% RSLogix 500 project DIGITAL_CONTROL_LOGIC.RSS, saved by version 8.30.00.16 %
PROJECT "DCL_L2P1"    % processor: Bul.1763 MicroLogix 1100 Series B %

PROGRAM FILES
  LAD 2 "MAIN"  5 rungs
  LAD 3 "DIGI IN"  3 rungs
  LAD 4 "DIGI OUT"  3 rungs
  LAD 5 "CONTROL"  7 rungs

DATA FILES
  O0 OUTPUT  5 elements
  I1 INPUT  7 elements
  S2 STATUS  66 elements
  B3 BINARY  3 elements
  T4 TIMER  4 elements
  C5 COUNTER  1 elements
  R6 CONTROL  1 elements
  N7 INTEGER  2 elements
  F8 FLOAT  1 elements

LADDER 2 "MAIN"
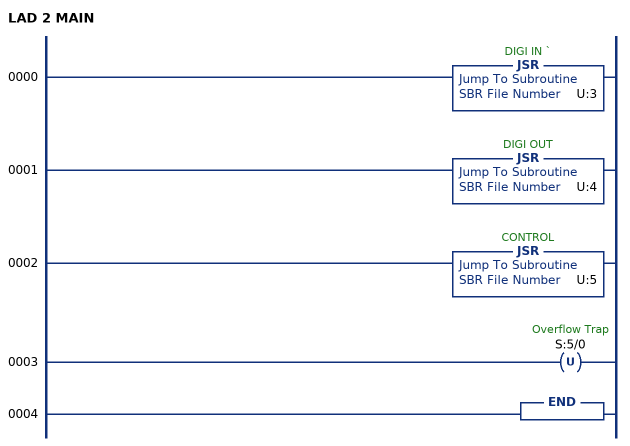
% Rung: 0 %
SOR JSR U:3 EOR
%   U:3  "DIGI IN `" %
% Rung: 1 %
SOR JSR U:4 EOR
%   U:4  "DIGI OUT" %
% Rung: 2 %
SOR JSR U:5 EOR
%   U:5  "CONTROL" %
% Rung: 3 %
SOR OTU S:5/0 EOR
%   S:5/0  "Overflow Trap" %
% Rung: 4 %
SOR END EOR

LADDER 3 "DIGI IN"
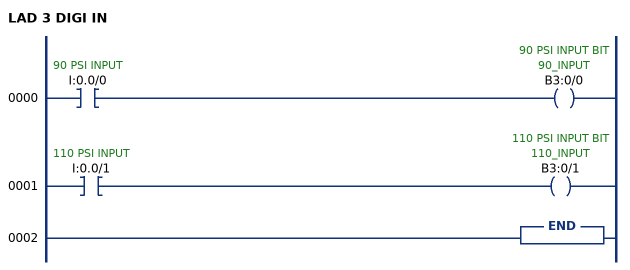
% Rung: 0 %
SOR XIC I:0.0/0 OTE B3:0/0 EOR
%   I:0.0/0  "90 PSI INPUT" %
%   B3:0/0  90_INPUT  "90 PSI INPUT BIT" %
% Rung: 1 %
SOR XIC I:0.0/1 OTE B3:0/1 EOR
%   I:0.0/1  "110 PSI INPUT" %
%   B3:0/1  110_INPUT  "110 PSI INPUT BIT" %
% Rung: 2 %
SOR END EOR

LADDER 4 "DIGI OUT"
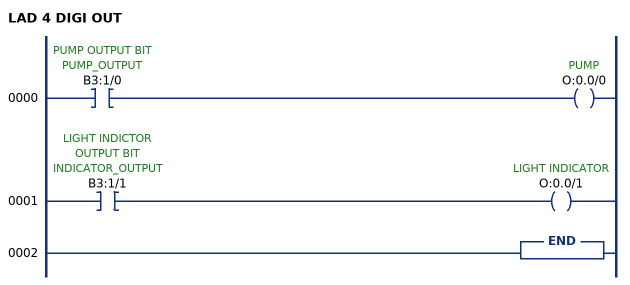
% Rung: 0 %
SOR XIC B3:1/0 OTE O:0.0/0 EOR
%   B3:1/0  PUMP_OUTPUT  "PUMP OUTPUT BIT" %
%   O:0.0/0  "PUMP" %
% Rung: 1 %
SOR XIC B3:1/1 OTE O:0.0/1 EOR
%   B3:1/1  INDICATOR_OUTPUT  "LIGHT INDICTOR OUTPUT BIT" %
%   O:0.0/1  "LIGHT INDICATOR" %
% Rung: 2 %
SOR END EOR

LADDER 5 "CONTROL"
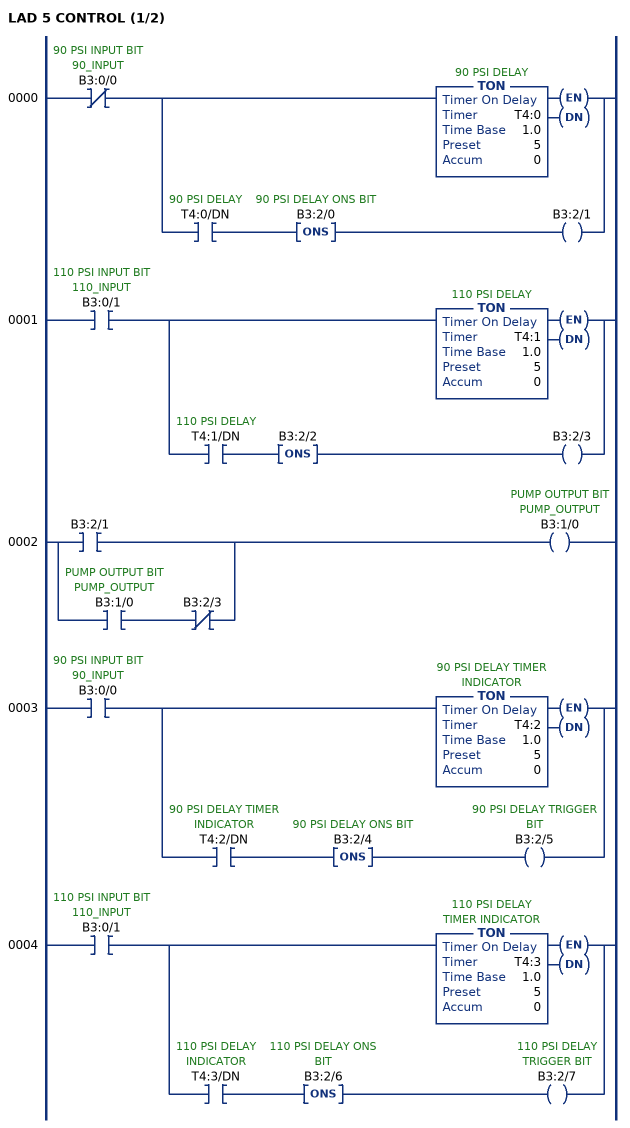
% Rung: 0 %
SOR XIO B3:0/0 BST TON T4:0 1.0 5 0 NXB XIC T4:0/DN ONS B3:2/0 OTE B3:2/1 BND EOR
%   B3:0/0  90_INPUT  "90 PSI INPUT BIT" %
%   T4:0  "90 PSI DELAY" %
%   T4:0/DN  "90 PSI DELAY" %
%   B3:2/0  "90 PSI DELAY ONS BIT" %
% Rung: 1 %
SOR XIC B3:0/1 BST TON T4:1 1.0 5 0 NXB XIC T4:1/DN ONS B3:2/2 OTE B3:2/3 BND EOR
%   B3:0/1  110_INPUT  "110 PSI INPUT BIT" %
%   T4:1  "110 PSI DELAY" %
% Rung: 2 %
SOR BST XIC B3:2/1 NXB XIC B3:1/0 XIO B3:2/3 BND OTE B3:1/0 EOR
%   B3:1/0  PUMP_OUTPUT  "PUMP OUTPUT BIT" %
% Rung: 3 %
SOR XIC B3:0/0 BST TON T4:2 1.0 5 0 NXB XIC T4:2/DN ONS B3:2/4 OTE B3:2/5 BND EOR
%   B3:0/0  90_INPUT  "90 PSI INPUT BIT" %
%   T4:2  "90 PSI DELAY TIMER INDICATOR" %
%   B3:2/4  "90 PSI DELAY ONS BIT" %
%   B3:2/5  "90 PSI DELAY TRIGGER BIT" %
% Rung: 4 %
SOR XIC B3:0/1 BST TON T4:3 1.0 5 0 NXB XIC T4:3/DN ONS B3:2/6 OTE B3:2/7 BND EOR
%   B3:0/1  110_INPUT  "110 PSI INPUT BIT" %
%   T4:3  "110 PSI DELAY TIMER INDICATOR" %
%   T4:3/DN  "110 PSI DELAY INDICATOR" %
%   B3:2/6  "110 PSI DELAY ONS BIT" %
%   B3:2/7  "110 PSI DELAY TRIGGER BIT" %

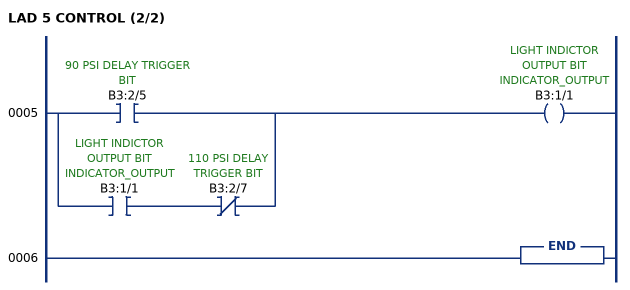
% Rung: 5 %  % edit flag set %
SOR BST XIC B3:2/5 NXB XIC B3:1/1 XIO B3:2/7 BND OTE B3:1/1 EOR
%   B3:2/5  "90 PSI DELAY TRIGGER BIT" %
%   B3:1/1  INDICATOR_OUTPUT  "LIGHT INDICTOR OUTPUT BIT" %
%   B3:2/7  "110 PSI DELAY TRIGGER BIT" %
% Rung: 6 %
SOR END EOR

OTHER DOCUMENTED ADDRESSES
  B2:0/0  "90 PSI DELAY ONS BIT"
  B2:2/0  "90 PSI DELAY ONS BIT"
  N7:0  PUMP_MODE  "PUMP MODE 0 = OFF 1 = ON"
  N7:1  INDICATOR_MODE  "INDICATOR MODE 0 = OFF 1 = ON"

DATA TABLE (non-zero values as saved)
DATA T4
% .PRE .ACC %
% T4:0 % 5 0
% T4:1 % 5 0
% T4:2 % 5 0
% T4:3 % 5 0
